// Mitsubishi GX Works2 project: 230930-001- exercicios-0   PLC: Q03UDV

// task Task_01 (event TRUE, interval 0, priority 31): POU_01

PROGRAM POU_01
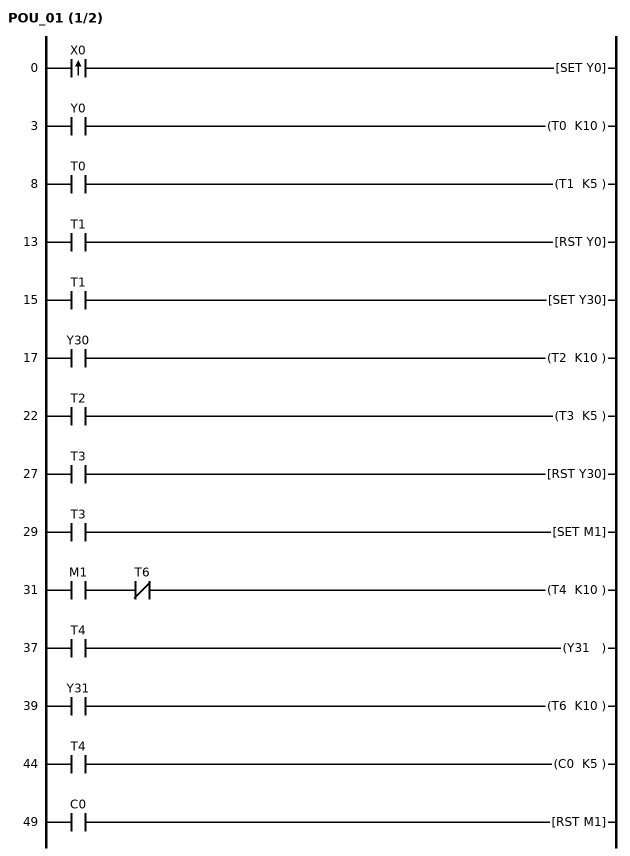
0     LDP     X0
      SET     Y0
3     LD      Y0
      OUT     T0 K10
8     LD      T0
      OUT     T1 K5
13    LD      T1
      RST     Y0
15    LD      T1
      SET     Y30
17    LD      Y30
      OUT     T2 K10
22    LD      T2
      OUT     T3 K5
27    LD      T3
      RST     Y30
29    LD      T3
      SET     M1
31    LD      M1
      ANI     T6
      OUT     T4 K10
37    LD      T4
      OUT     Y31
39    LD      Y31
      OUT     T6 K10
44    LD      T4
      OUT     C0 K5
49    LD      C0
      RST     M1
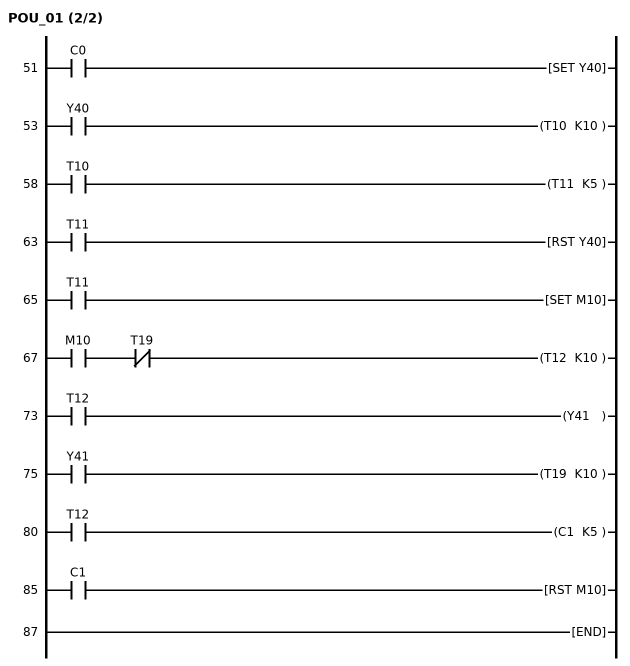
51    LD      C0
      SET     Y40
53    LD      Y40
      OUT     T10 K10
58    LD      T10
      OUT     T11 K5
63    LD      T11
      RST     Y40
65    LD      T11
      SET     M10
67    LD      M10
      ANI     T19
      OUT     T12 K10
73    LD      T12
      OUT     Y41
75    LD      Y41
      OUT     T19 K10
80    LD      T12
      OUT     C1 K5
85    LD      C1
      RST     M10
87    END
END_PROGRAM
